Staubli VAL3: selectType.pgx

program selectType(string& x_sItem)
  local num l_nSizeList
  local string l_sItem
  local bool l_bActive
  local string l_sItemList
  local string l_sMessage
  local num l_nKey
  local string l_sEvent
  local num l_nSize
  local num i
  local string l_sName
begin
  // CNT
  call saveInOut:getSize_num(l_nSizeList)
  call getType(l_sItem)
  l_nSize=0
  //
  // create the list
  //
  call use:setSizeList(19,0,19,11)
  call use:listcreate(l_sItem)
  // insert in the list
  for i=0 to l_nSizeList-1
    call saveInOut:get_num(l_sItemList,i)
    call isActive(l_bActive,l_sItemList)
    if l_bActive
      call saveInOut:get_num(l_sItemList,i)
      call saveInOut:getItem_num(l_sName,l_sItemList)
      l_sItemList=l_sItemList+" {"+l_sName+"}"
      call use:listadd(l_sItemList)
    endIf
  endFor
  call use:selectNewField(nIndex,nIndex,0)
  call use:clear(0,13)
  call language:message(l_sMessage,63)
  call use:typeCenter(13,l_sMessage,40,true)
  do
    // get the key
    l_nKey=get()
    // get one input from the list
    call use:listevent(l_nKey,nIndex,l_sEvent)
    if l_nKey==255
      return
    endIf
  until l_nKey==270
  // save it
  if l_sEvent!=""
    x_sItem=left(l_sEvent,find(l_sEvent,"{")-1)
  else
    x_sItem=""
  endIf
end
